{attribute 'linkalways'} 
{attribute 'no_explicit_call' := 'This FB is a CLASS and must be accessed using methods or properties'}
{attribute 'enable_dynamic_creation'}
FUNCTION_BLOCK Node_F_VN_FillContainer_TcVnKeyPoint EXTENDS VisionNode
VAR
    ipContainer : _ITcVnContainer;
    stValue : _TcVnKeyPoint;
    hrPrev : _HRESULT(S_OK);
    hresult : _HRESULT(S_OK);
END_VAR

METHOD PUBLIC  Clone : I_Node
VAR
    pNode : POINTER TO Node_F_VN_FillContainer_TcVnKeyPoint;
END_VAR
pNode := __NEW(Node_F_VN_FillContainer_TcVnKeyPoint);
Clone := pNode^;
END_METHOD

METHOD FB_init : BOOL
VAR_INPUT
    bInitRetains : BOOL; // if TRUE, the retain variables are initialized (warm start / cold start)
    bInCopyCode : BOOL;  // if TRUE, the instance afterwards gets moved into the copy code (online change)
END_VAR
AddInput('ipContainer', ipContainer);
AddInput('stValue', stValue);
AddInput('hrPrev', hrPrev);
AddOutput('ipContainer', ipContainer);
AddOutput('hresult',hresult);
END_METHOD

METHOD PROTECTED OnExecute : HRESULT
hresult.Value := F_VN_FillContainer_TcVnKeyPoint(
    ipContainer := ipContainer.Value,
    stValue := stValue.Value,
    hrPrev:= hrPrev.Value);
END_METHOD

METHOD PUBLIC PreExecutionCheck
VAR_INPUT
    Check : I_PreExecutionChecks;
END_VAR
Check.IsTrue(ipContainer.IsValid, 'ipContainer must be a valid container');
END_METHOD

END_FUNCTION_BLOCK

(* stored: Version 1.1.0.1, ProductVersion 3.1.4024.13
   POU Node_F_VN_FillContainer_TcVnKeyPoint: Id {9a2bea6c-1b42-484f-8d62-c8e63f1d211b}, SpecialFunc None
   Folder Constructor: Id {1ec4c1d7-66bb-4570-8abf-b83f0c0ec2b4}
   Method Clone: Id {034a51b0-c3c5-4bcc-9242-38b7a4dab892}
   Method FB_init: Id {45737944-4f03-455e-8b95-f26b79ce1e19}
   Method OnExecute: Id {2689206b-7e75-4dc4-a589-bf16d76c8b82}
   Method PreExecutionCheck: Id {2d1c57b9-d820-479c-9138-c4932dd5a03f} *)
